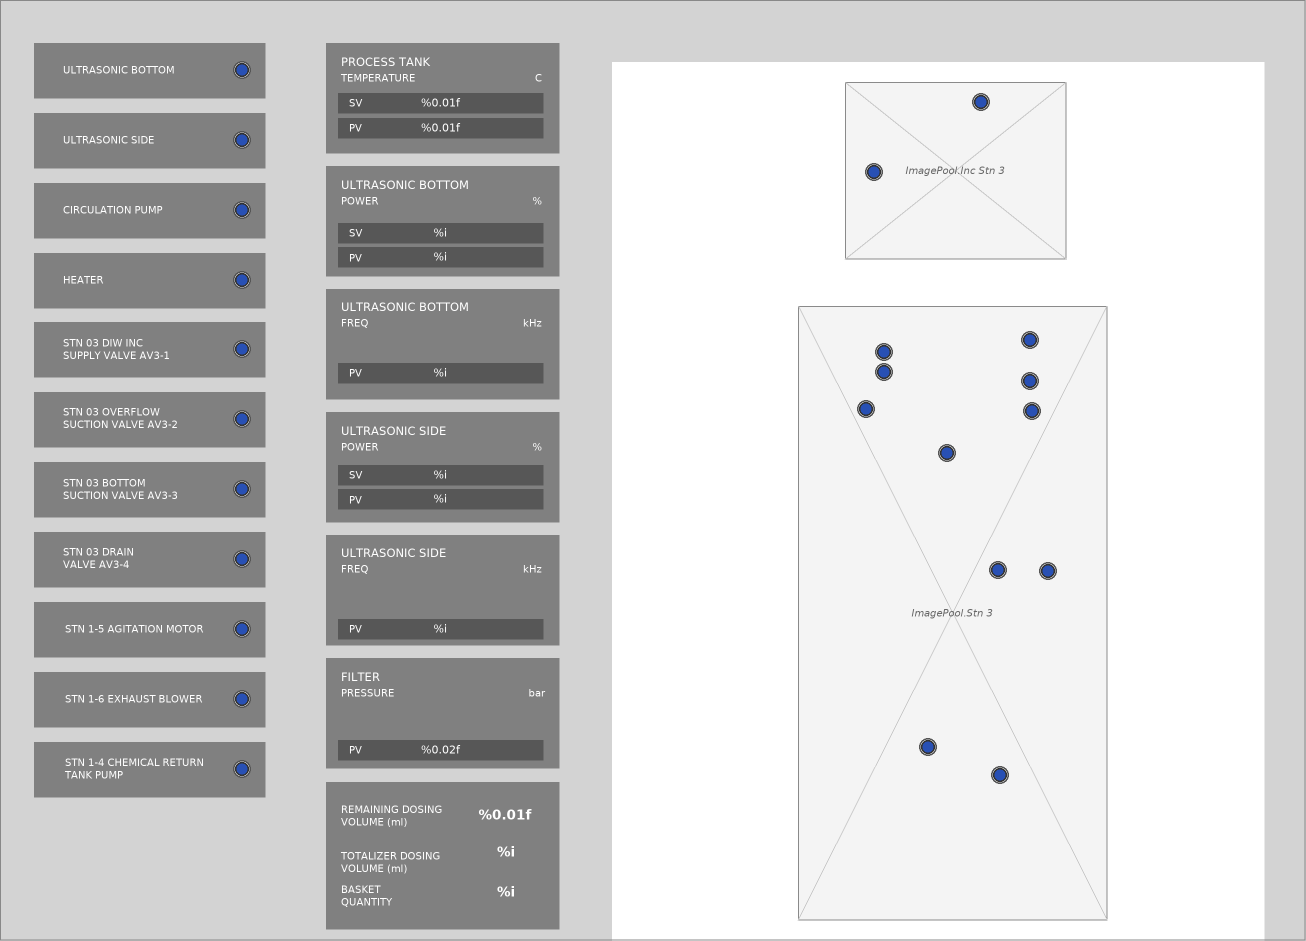
VISUALIZATION Auto_Station03  // 1306x941
    Rectangle (0,0 1306x875)
    RoundedRectangle (34,43 231x55)
    Label (60,62 163x16), "ULTRASONIC BOTTOM"
    Lamp1 (232,60 20x20), variable: ARdsMAP_HmiVariableStn[3].bProTankUsBtm_IND, style: Lamp-Lamp1-Blue
    RoundedRectangle (34,183 231x55)
    Label (60,202 151x16), "CIRCULATION PUMP"
    Lamp1 (232,200 20x20), variable: ARdsMAP_HmiVariableStn[3].bProTankPump_IND, style: Lamp-Lamp1-Blue
    RoundedRectangle (34,253 231x55)
    Label (60,272 151x16), "HEATER"
    Lamp1 (232,270 20x20), variable: ARdsMAP_HmiVariableStn[3].bProTankHeater_IND, style: Lamp-Lamp1-Blue
    RoundedRectangle (34,113 231x55)
    Label (60,132 163x16), "ULTRASONIC SIDE"
    Lamp1 (232,130 20x20), variable: ARdsMAP_HmiVariableStn[3].bProTankUsSide_IND, style: Lamp-Lamp1-Blue
    RoundedRectangle (34,322 231x55)
    Label (60,336 151x27), "STN 03 DIW INC SUPPLY VALVE AV3-1"
    Lamp1 (232,339 20x20), variable: ARdsMAP_HmiVariableStn[3].bValve01_IND, style: Lamp-Lamp1-Blue
    RoundedRectangle (34,392 231x55)
    Lamp1 (232,409 20x20), variable: ARdsMAP_HmiVariableStn[3].bValve02_IND, style: Lamp-Lamp1-Blue
    Label (60,405 168x27), "STN 03 OVERFLOW SUCTION VALVE AV3-2"
    RoundedRectangle (34,462 231x55)
    Label (60,476 151x27), "STN 03 BOTTOM SUCTION VALVE AV3-3"
    Lamp1 (232,479 20x20), variable: ARdsMAP_HmiVariableStn[3].bValve03_IND, style: Lamp-Lamp1-Blue
    RoundedRectangle (34,532 231x55)
    Lamp1 (232,549 20x20), variable: ARdsMAP_HmiVariableStn[3].bValve04_IND, style: Lamp-Lamp1-Blue
    Label (60,545 168x27), "STN 03 DRAIN VALVE AV3-4"
    RoundedRectangle (34,602 231x55)
    Label (62,611 160x36), "STN 1-5 AGITATION MOTOR"
    Lamp1 (232,619 20x20), variable: ARdsMAP_HmiVariableGeneral.bProTankAgitationMotor_IND, style: Lamp-Lamp1-Blue
    RoundedRectangle (34,672 231x55)
    Label (62,681 160x36), "STN 1-6 EXHAUST BLOWER"
    Lamp1 (232,689 20x20), variable: ARdsMAP_HmiVariableGeneral.bExhaustBlower_IND, style: Lamp-Lamp1-Blue
    RoundedRectangle (34,742 231x55)
    Label (62,751 160x36), "STN 1-4 CHEMICAL RETURN TANK PUMP"
    Lamp1 (232,759 20x20), variable: ARdsMAP_HmiVariableGeneral.bProTankPump_IND, style: Lamp-Lamp1-Blue
    Rectangle (612,62 652x879)
    Image (798,306 309x614), image: ImagePool.Stn 3
    Lamp1 (937,443 20x20), variable: ARdsMAP_HmiVariableStn[3].bProTankUsBtm_IND, style: Lamp-Lamp1-Blue
    Lamp1 (918,737 20x20), variable: ARdsMAP_HmiVariableStn[3].bProTankPump_IND, style: Lamp-Lamp1-Blue
    Lamp1 (874,362 20x20), variable: ARdsMAP_HmiVariableStn[3].bProTankHeater_IND, style: Lamp-Lamp1-Blue
    Lamp1 (856,399 20x20), variable: ARdsMAP_HmiVariableStn[3].bProTankUsSide_IND, style: Lamp-Lamp1-Blue
    Lamp1 (1038,561 20x20), variable: ARdsMAP_HmiVariableStn[3].bValve02_IND, style: Lamp-Lamp1-Blue
    Lamp1 (990,765 20x20), variable: ARdsMAP_HmiVariableStn[3].bValve04_IND, style: Lamp-Lamp1-Blue
    Lamp1 (988,560 20x20), variable: ARdsMAP_HmiVariableStn[3].bValve03_IND, style: Lamp-Lamp1-Blue
    Lamp1 (1020,330 20x20), variable: ARdsMAP_HmiVariableStn[3].bOverflowMaxLevel_IND, style: Lamp-Lamp1-Blue
    Lamp1 (874,342 20x20), variable: ARdsMAP_HmiVariableStn[3].bProcessTankMinLevel_IND, style: Lamp-Lamp1-Blue
    Lamp1 (1020,371 20x20), variable: ARdsMAP_HmiVariableStn[3].bOverflowMinLevel_IND, style: Lamp-Lamp1-Blue
    Lamp1 (1022,401 20x20), variable: ARdsMAP_HmiVariableStn[3].bProTankUsSide_IND, style: Lamp-Lamp1-Blue
    Image (845,82 221x177), image: ImagePool.Inc Stn 3
    Lamp1 (971,92 20x20), variable: ARdsMAP_HmiVariableStn[3].bValve01_IND, style: Lamp-Lamp1-Blue
    Lamp1 (864,162 20x20), variable: ARdsMAP_HmiVariableStn[3].bDosingPump_IND, style: Lamp-Lamp1-Blue
    RoundedRectangle (326,43 233x110)
    Label (338,54 150x16), "PROCESS TANK"
    Label (338,67 99x22), "TEMPERATURE"
    Label (516,67 29x22), "C"
    Rectangle (338,93 205x20), "%0.01f", text variable: ARrStnTempSV[3]
    Label (346,92 22x22), "SV"
    Rectangle (338,118 205x20), "%0.01f", text variable: ARrStnTempPV[3]
    Label (346,117 22x22), "PV"
    RoundedRectangle (326,166 233x110)
    Label (338,177 150x16), "ULTRASONIC BOTTOM"
    Label (338,190 99x22), "POWER"
    Label (516,190 29x22), "%"
    Rectangle (338,223 205x20), "%i", text variable: DSWeberEnclosure[1].DSWeberGenerator[6].IN_iTargetPowerPercentSetPoint
    Label (346,222 22x22), "SV"
    Rectangle (338,247 205x20), "%i", text variable: ARiStnUSBtmAPv[3]
    Label (346,247 22x22), "PV"
    RoundedRectangle (326,658 233x110)
    Label (338,669 150x16), "FILTER"
    Label (338,682 99x22), "PRESSURE"
    Label (516,682 32x22), "bar"
    Rectangle (338,740 205x20), "%0.02f", text variable: ARrStnFilterPressurePV[3]
    Label (346,739 22x22), "PV"
    RoundedRectangle (326,289 233x110)
    Label (338,312 99x22), "FREQ"
    Label (338,299 150x16), "ULTRASONIC BOTTOM"
    Label (516,312 29x22), "kHz"
    Rectangle (338,363 205x20), "%i", text variable: ARiStnUSBtmAFreqPv[3]
    Label (346,362 22x22), "PV"
    RoundedRectangle (326,782 233x147)
    Label (338,845 118x35), "TOTALIZER DOSING VOLUME (ml)"
    Label (338,802 118x28), "REMAINING DOSING VOLUME (ml)"
    Rectangle (464,801 82x28), "%0.01f", text variable: ARDSProminentDosingHMI[3].Out_rRemainedDosingVolume_ml
    Rectangle (465,838 82x28), "%i", text variable: ARDSProminentDosingHMI[3].Out_iDosingTotalizer_ml
    Label (338,882 118x28), "BASKET QUANTITY"
    Rectangle (465,878 82x28), "%i", text variable: ARDSProminentDosingHMI[3].Out_iBasketQtyBeforeAutoDosingPV
    RoundedRectangle (326,412 233x110)
    Label (338,423 150x16), "ULTRASONIC SIDE"
    Label (338,436 99x22), "POWER"
    Label (516,436 29x22), "%"
    Rectangle (338,465 205x20), "%i", text variable: DSWeberEnclosure[1].DSWeberGenerator[6].IN_iTargetPowerPercentSetPoint
    Label (346,464 22x22), "SV"
    Rectangle (338,489 205x20), "%i", text variable: ARiStnUSSideAPv[3]
    Label (346,489 22x22), "PV"
    RoundedRectangle (326,535 233x110)
    Label (338,558 99x22), "FREQ"
    Label (338,545 150x16), "ULTRASONIC SIDE"
    Label (516,558 29x22), "kHz"
    Rectangle (338,619 205x20), "%i", text variable: ARiStnUSSideAFreqPv[3]
    Label (346,618 22x22), "PV"
END_VISUALIZATION

(* stored: Version 1.1.0.1, ProductVersion 3.1.4024.12
   Visu Auto_Station03: Id {0a4d763d-8f58-4042-a8fa-50c3d3d723a3} *)
